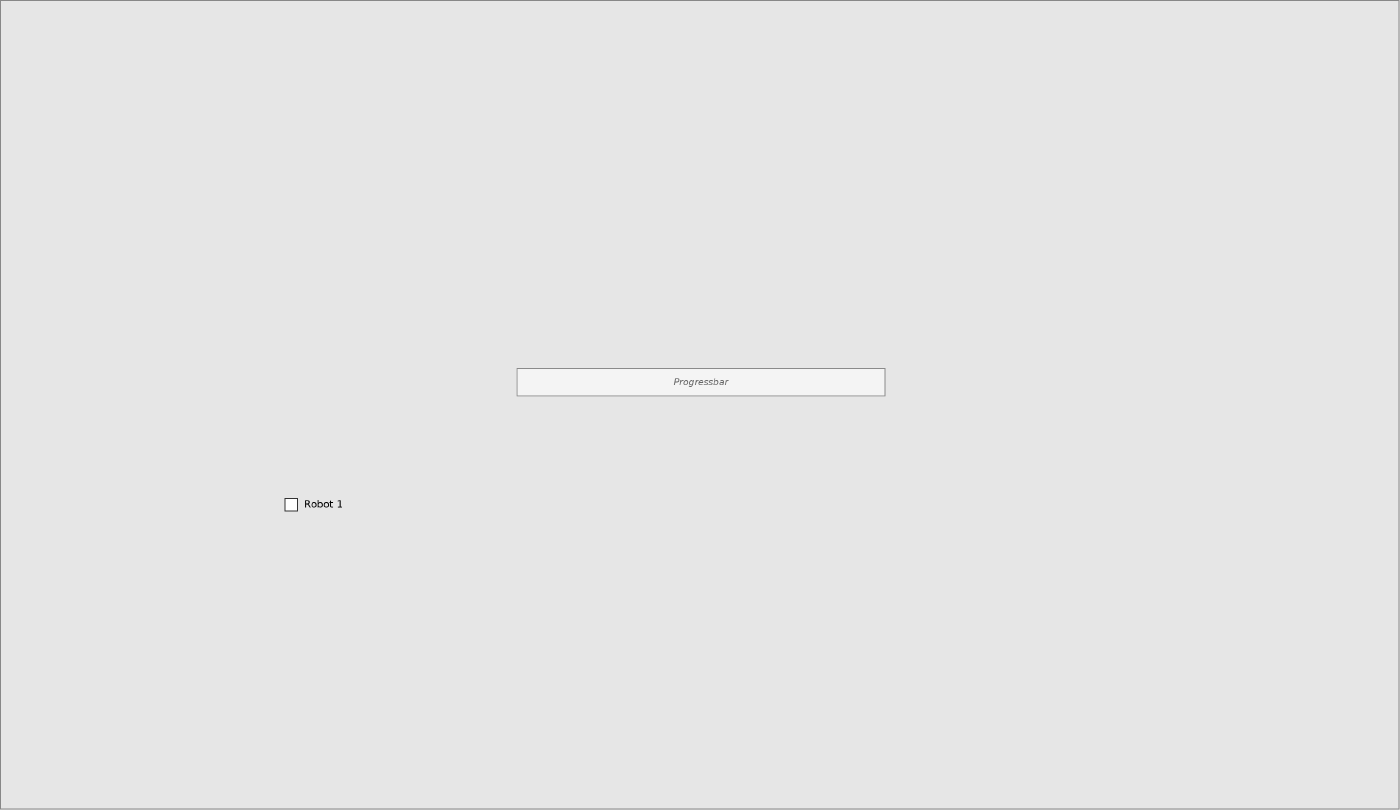
VISUALIZATION PageInitializing  // 1520x880
    Progressbar (561,400 400x30)
    Checkbox (307,533 320x30), "Robot 1"
END_VISUALIZATION

(* stored: Version 1.1.0.1, ProductVersion 3.1.4024.9
   Visu PageInitializing: Id {461aef6d-9bf3-405f-b92f-526b7bdc38b8} *)
